// TIA Portal V18 export
DATA_BLOCK "Initial_Test_Squence_DB"   // DB78
VERSION : 0.1
// stored: AutoNumber true, DBAccessibleFromOPCUA true, InstanceOfName Initial_Test_Squence, InstanceOfType FB
"Initial_Test_Squence"
   // VAR_INPUT
   //    ON : Bool;
   //    Position : DInt;
   //    HomingOK : Bool;
   //    InputTask : Bool;
   //    StepSizeInput : DInt;
   //    AmountOfSteps : Int;
   // END_VAR
   // VAR_OUTPUT
   //    StartMachine : Bool;
   //    StartHoming : Bool;
   //    StepSizeOutput : DInt;
   //    TestFinished : Bool;
   //    StartPosition : DInt;
   //    EndPositon : DInt;
   // END_VAR
   // VAR_IN_OUT
   //    StartTask : Bool;
   // END_VAR
   // VAR
   //    TurnOnM : Bool;
   //    StepNumber : Int;
   //    InternalWait { ExternalAccessible := 'False'; ExternalVisible := 'False'; ExternalWritable := 'False'} : Bool;
   //    StepNumberNext { ExternalAccessible := 'False'; ExternalVisible := 'False'; ExternalWritable := 'False'} : Int;
   //    ONM : Bool;
   //    TestFinishedM : Bool;
   //    StartTaskM { ExternalAccessible := 'False'; ExternalVisible := 'False'; ExternalWritable := 'False'} : Bool;
   // END_VAR
BEGIN
END_DATA_BLOCK
